FUNCTION_BLOCK HCylAdp (* Composite Function Block Type *)
  (* Standard: 61499-2 *)
  (* Version 0.0, 06/10/2018, Atmojo, nxtControl GmbH, template *)
  PACKAGE Main;
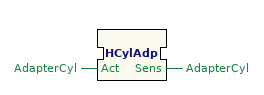
  SOCKETS
    Act : AdapterCyl;
  END_SOCKETS
  PLUGS
    Sens : AdapterCyl;
  END_PLUGS
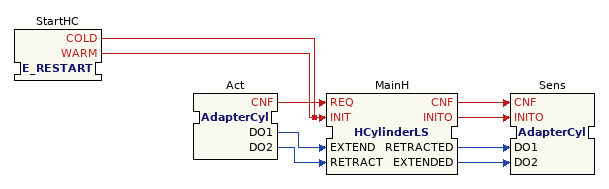
  FBS
    MainH : HCylinderLS;
    StartHC : E_RESTART;
  END_FBS
  EVENT_CONNECTIONS
    Act.CNF TO MainH.REQ;
    MainH.CNF TO Sens.CNF;
    MainH.INITO TO Sens.INITO;
    StartHC.COLD TO MainH.INIT;
    StartHC.WARM TO MainH.INIT;
  END_CONNECTIONS
  DATA_CONNECTIONS
    Act.DO1 TO MainH.EXTEND;
    Act.DO2 TO MainH.RETRACT;
    MainH.RETRACTED TO Sens.DO1;
    MainH.EXTENDED TO Sens.DO2;
  END_CONNECTIONS
END_FUNCTION_BLOCK
